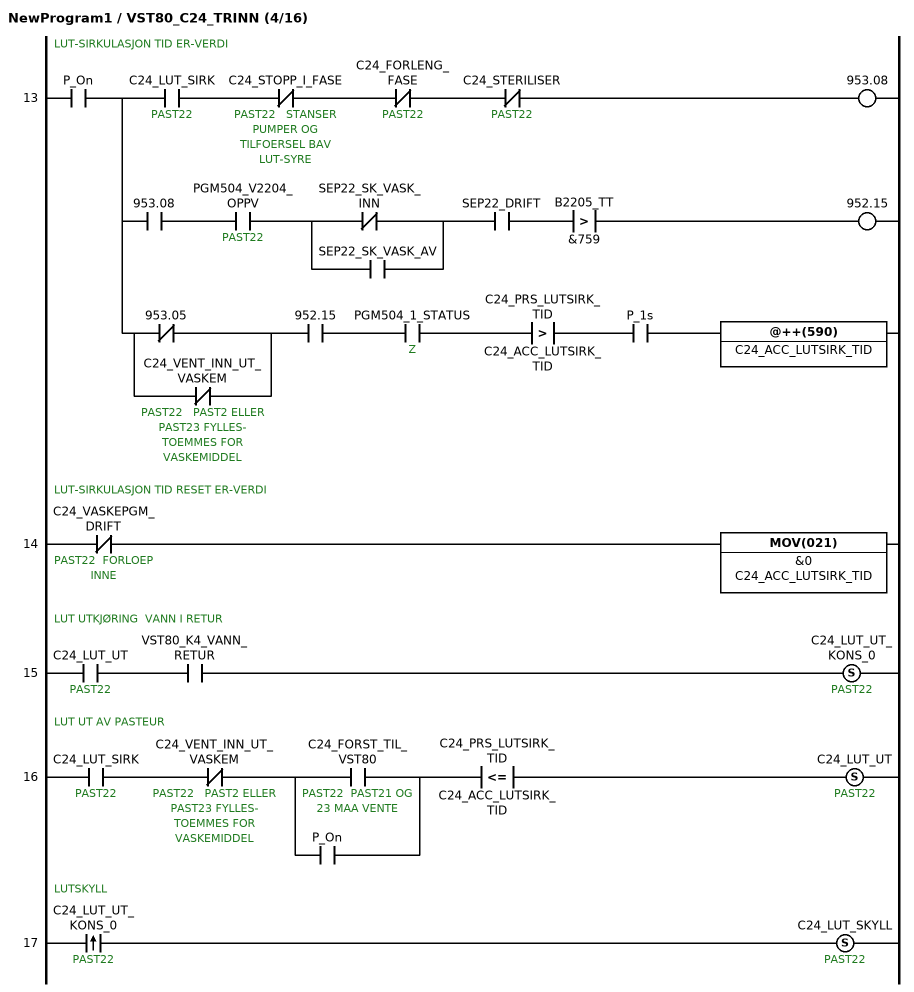
; [picture p432: NewProgram1 / VST80_C24_TRINN, rungs 13-17]
; rung 13: LUT-SIRKULASJON TID ER-VERDI
LD P_On
OUT TR0
AND C24_LUT_SIRK  ; PAST22
ANDNOT C24_STOPP_I_FASE  ; PAST22   STANSER PUMPER OG TILFOERSEL BAV LUT-SYRE
ANDNOT C24_FORLENG_FASE  ; PAST22
ANDNOT C24_STERILISER  ; PAST22
OUT 953.08
LD TR0
AND 953.08
AND PGM504_V2204_OPPV  ; PAST22
LDNOT SEP22_SK_VASK_INN
OR SEP22_SK_VASK_AV
ANDLD
AND SEP22_DRIFT
AND>(320) B2205_TT &759
OUT 952.15
LD TR0
LDNOT 953.05
ORNOT C24_VENT_INN_UT_VASKEM  ; PAST22   PAST2 ELLER PAST23 FYLLES-TOEMMES FOR VASKEMIDDEL
ANDLD
AND 952.15
AND PGM504_1_STATUS  ; Z
AND>(320) C24_PRS_LUTSIRK_TID C24_ACC_LUTSIRK_TID
AND P_1s
@++(590) C24_ACC_LUTSIRK_TID
; rung 14: LUT-SIRKULASJON TID RESET ER-VERDI
LDNOT C24_VASKEPGM_DRIFT  ; PAST22  FORLOEP INNE
MOV(021) &0 C24_ACC_LUTSIRK_TID
; rung 15: LUT UTKJØRING  VANN I RETUR
LD C24_LUT_UT  ; PAST22
AND VST80_K4_VANN_RETUR
SET C24_LUT_UT_KONS_0  ; PAST22
; rung 16: LUT UT AV PASTEUR
LD C24_LUT_SIRK  ; PAST22
ANDNOT C24_VENT_INN_UT_VASKEM  ; PAST22   PAST2 ELLER PAST23 FYLLES-TOEMMES FOR VASKEMIDDEL
LD C24_FORST_TIL_VST80  ; PAST22  PAST21 OG 23 MAA VENTE
OR P_On
ANDLD
AND<=(315) C24_PRS_LUTSIRK_TID C24_ACC_LUTSIRK_TID
SET C24_LUT_UT  ; PAST22
; rung 17: LUTSKYLL
@LD C24_LUT_UT_KONS_0  ; PAST22
SET C24_LUT_SKYLL  ; PAST22

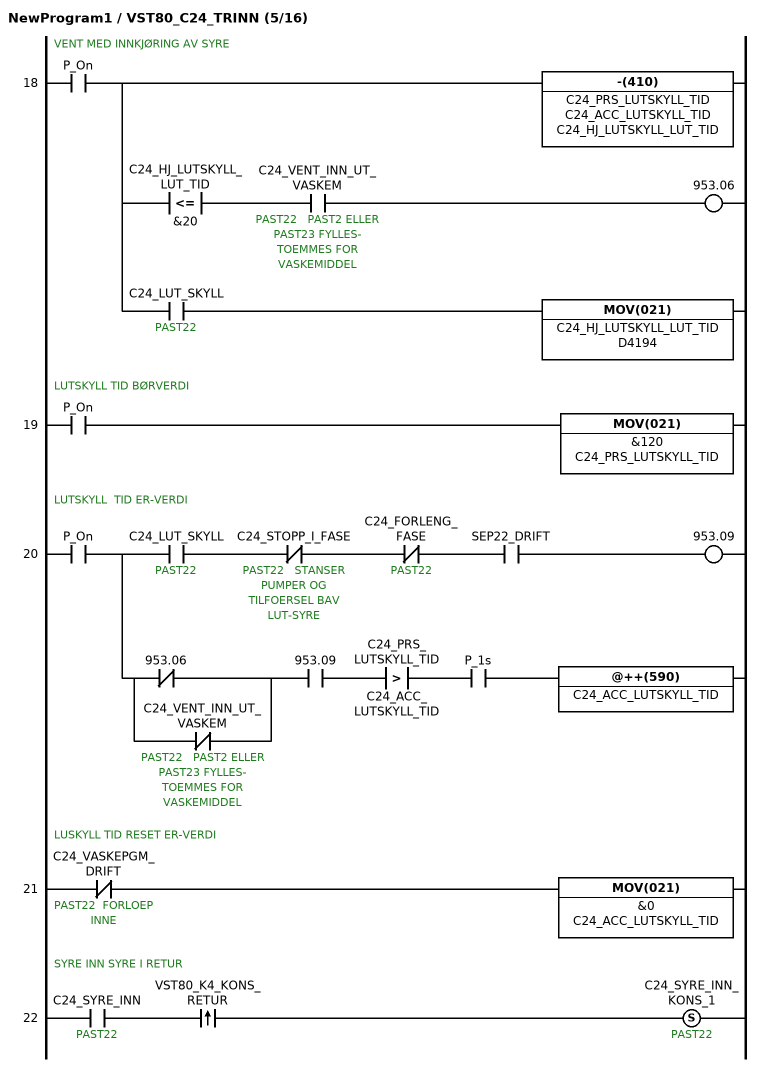
; rung 18: VENT MED INNKJØRING AV SYRE
LD P_On
OUT TR0
-(410) C24_PRS_LUTSKYLL_TID C24_ACC_LUTSKYLL_TID C24_HJ_LUTSKYLL_LUT_TID
AND<=(315) C24_HJ_LUTSKYLL_LUT_TID &20
AND C24_VENT_INN_UT_VASKEM  ; PAST22   PAST2 ELLER PAST23 FYLLES-TOEMMES FOR VASKEMIDDEL
OUT 953.06
LD TR0
AND C24_LUT_SKYLL  ; PAST22
MOV(021) C24_HJ_LUTSKYLL_LUT_TID D4194
; rung 19: LUTSKYLL TID BØRVERDI
LD P_On
MOV(021) &120 C24_PRS_LUTSKYLL_TID
; rung 20: LUTSKYLL  TID ER-VERDI
LD P_On
OUT TR0
AND C24_LUT_SKYLL  ; PAST22
ANDNOT C24_STOPP_I_FASE  ; PAST22   STANSER PUMPER OG TILFOERSEL BAV LUT-SYRE
ANDNOT C24_FORLENG_FASE  ; PAST22
AND SEP22_DRIFT
OUT 953.09
LD TR0
LDNOT 953.06
ORNOT C24_VENT_INN_UT_VASKEM  ; PAST22   PAST2 ELLER PAST23 FYLLES-TOEMMES FOR VASKEMIDDEL
ANDLD
AND 953.09
AND>(320) C24_PRS_LUTSKYLL_TID C24_ACC_LUTSKYLL_TID
AND P_1s
@++(590) C24_ACC_LUTSKYLL_TID
; rung 21: LUSKYLL TID RESET ER-VERDI
LDNOT C24_VASKEPGM_DRIFT  ; PAST22  FORLOEP INNE
MOV(021) &0 C24_ACC_LUTSKYLL_TID
; rung 22: SYRE INN SYRE I RETUR
LD C24_SYRE_INN  ; PAST22
@AND VST80_K4_KONS_RETUR
SET C24_SYRE_INN_KONS_1  ; PAST22

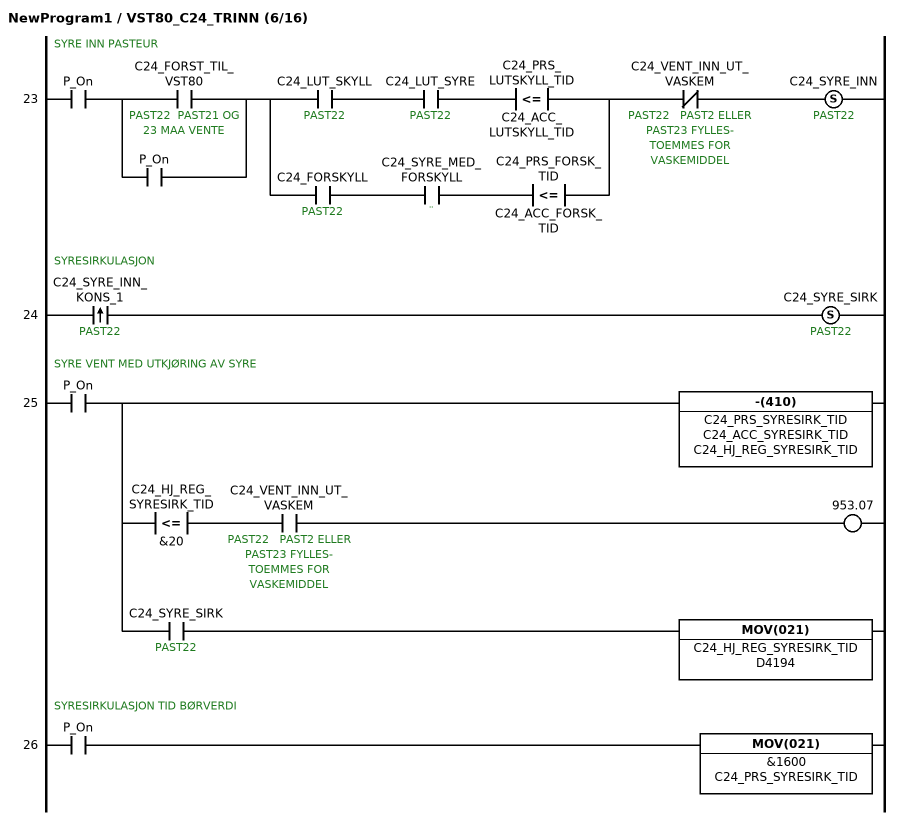
; rung 23: SYRE INN PASTEUR
LD P_On
LD C24_FORST_TIL_VST80  ; PAST22  PAST21 OG 23 MAA VENTE
OR P_On
ANDLD
LD C24_LUT_SKYLL  ; PAST22
AND C24_LUT_SYRE  ; PAST22
AND<=(315) C24_PRS_LUTSKYLL_TID C24_ACC_LUTSKYLL_TID
LD C24_FORSKYLL  ; PAST22
AND C24_SYRE_MED_FORSKYLL  ; ¨
AND<=(315) C24_PRS_FORSK_TID C24_ACC_FORSK_TID
ORLD
ANDLD
ANDNOT C24_VENT_INN_UT_VASKEM  ; PAST22   PAST2 ELLER PAST23 FYLLES-TOEMMES FOR VASKEMIDDEL
SET C24_SYRE_INN  ; PAST22
; rung 24: SYRESIRKULASJON
@LD C24_SYRE_INN_KONS_1  ; PAST22
SET C24_SYRE_SIRK  ; PAST22
; rung 25: SYRE VENT MED UTKJØRING AV SYRE
LD P_On
OUT TR0
-(410) C24_PRS_SYRESIRK_TID C24_ACC_SYRESIRK_TID C24_HJ_REG_SYRESIRK_TID
AND<=(315) C24_HJ_REG_SYRESIRK_TID &20
AND C24_VENT_INN_UT_VASKEM  ; PAST22   PAST2 ELLER PAST23 FYLLES-TOEMMES FOR VASKEMIDDEL
OUT 953.07
LD TR0
AND C24_SYRE_SIRK  ; PAST22
MOV(021) C24_HJ_REG_SYRESIRK_TID D4194
; rung 26: SYRESIRKULASJON TID BØRVERDI
LD P_On
MOV(021) &1600 C24_PRS_SYRESIRK_TID

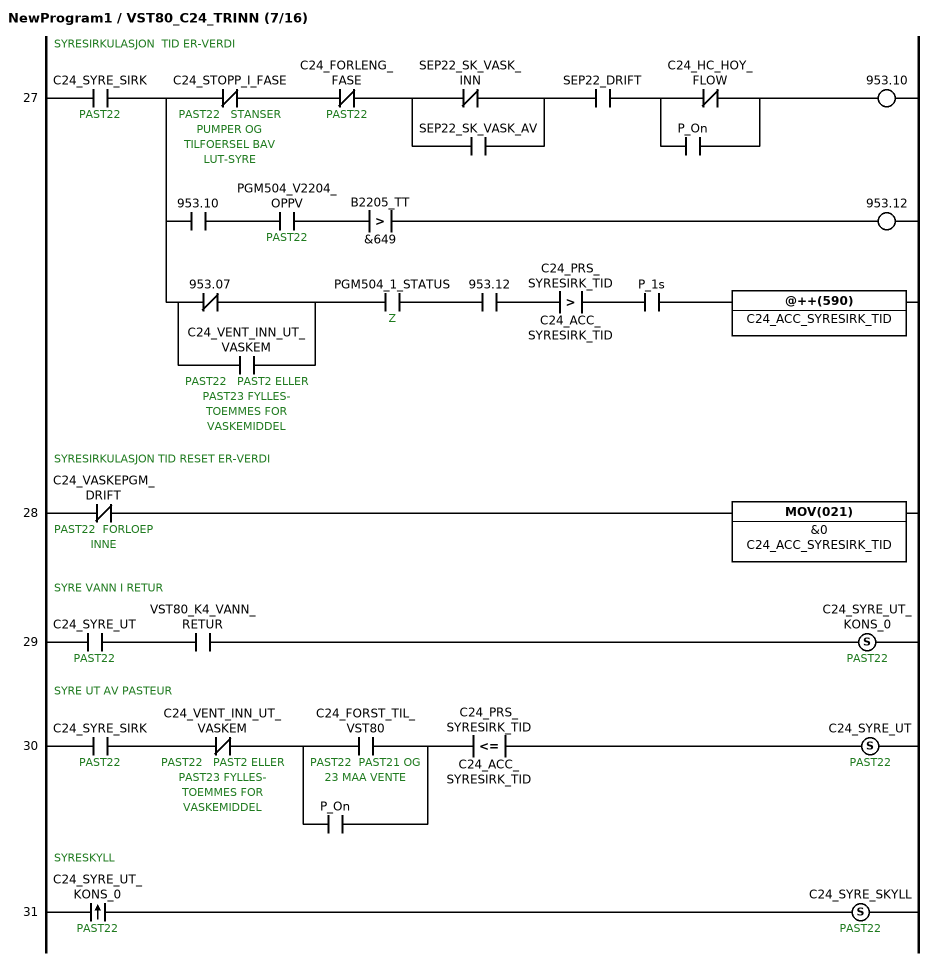
; rung 27: SYRESIRKULASJON  TID ER-VERDI
LD C24_SYRE_SIRK  ; PAST22
OUT TR0
ANDNOT C24_STOPP_I_FASE  ; PAST22   STANSER PUMPER OG TILFOERSEL BAV LUT-SYRE
ANDNOT C24_FORLENG_FASE  ; PAST22
LDNOT SEP22_SK_VASK_INN
OR SEP22_SK_VASK_AV
ANDLD
AND SEP22_DRIFT
LDNOT C24_HC_HOY_FLOW
OR P_On
ANDLD
OUT 953.10
LD TR0
AND 953.10
AND PGM504_V2204_OPPV  ; PAST22
AND>(320) B2205_TT &649
OUT 953.12
LD TR0
LDNOT 953.07
OR C24_VENT_INN_UT_VASKEM  ; PAST22   PAST2 ELLER PAST23 FYLLES-TOEMMES FOR VASKEMIDDEL
ANDLD
AND PGM504_1_STATUS  ; Z
AND 953.12
AND>(320) C24_PRS_SYRESIRK_TID C24_ACC_SYRESIRK_TID
AND P_1s
@++(590) C24_ACC_SYRESIRK_TID
; rung 28: SYRESIRKULASJON TID RESET ER-VERDI
LDNOT C24_VASKEPGM_DRIFT  ; PAST22  FORLOEP INNE
MOV(021) &0 C24_ACC_SYRESIRK_TID
; rung 29: SYRE VANN I RETUR
LD C24_SYRE_UT  ; PAST22
AND VST80_K4_VANN_RETUR
SET C24_SYRE_UT_KONS_0  ; PAST22
; rung 30: SYRE UT AV PASTEUR
LD C24_SYRE_SIRK  ; PAST22
ANDNOT C24_VENT_INN_UT_VASKEM  ; PAST22   PAST2 ELLER PAST23 FYLLES-TOEMMES FOR VASKEMIDDEL
LD C24_FORST_TIL_VST80  ; PAST22  PAST21 OG 23 MAA VENTE
OR P_On
ANDLD
AND<=(315) C24_PRS_SYRESIRK_TID C24_ACC_SYRESIRK_TID
SET C24_SYRE_UT  ; PAST22
; rung 31: SYRESKYLL
@LD C24_SYRE_UT_KONS_0  ; PAST22
SET C24_SYRE_SKYLL  ; PAST22

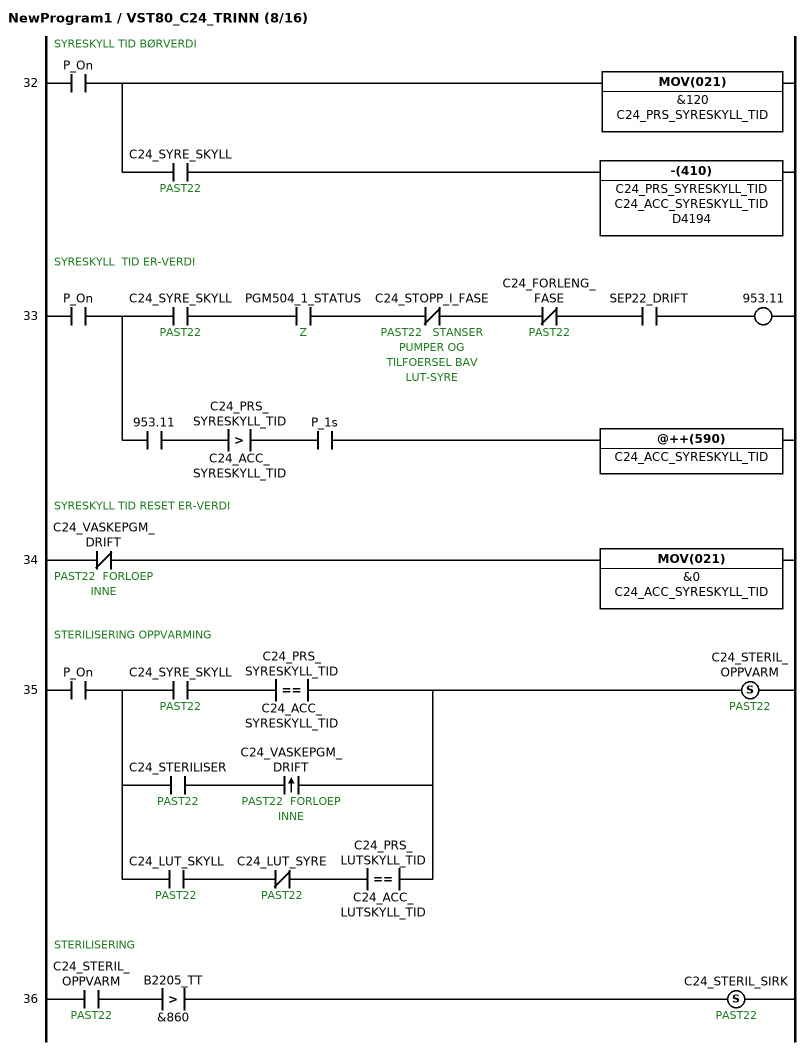
; rung 32: SYRESKYLL TID BØRVERDI
LD P_On
MOV(021) &120 C24_PRS_SYRESKYLL_TID
AND C24_SYRE_SKYLL  ; PAST22
-(410) C24_PRS_SYRESKYLL_TID C24_ACC_SYRESKYLL_TID D4194
; rung 33: SYRESKYLL  TID ER-VERDI
LD P_On
OUT TR0
AND C24_SYRE_SKYLL  ; PAST22
AND PGM504_1_STATUS  ; Z
ANDNOT C24_STOPP_I_FASE  ; PAST22   STANSER PUMPER OG TILFOERSEL BAV LUT-SYRE
ANDNOT C24_FORLENG_FASE  ; PAST22
AND SEP22_DRIFT
OUT 953.11
LD TR0
AND 953.11
AND>(320) C24_PRS_SYRESKYLL_TID C24_ACC_SYRESKYLL_TID
AND P_1s
@++(590) C24_ACC_SYRESKYLL_TID
; rung 34: SYRESKYLL TID RESET ER-VERDI
LDNOT C24_VASKEPGM_DRIFT  ; PAST22  FORLOEP INNE
MOV(021) &0 C24_ACC_SYRESKYLL_TID
; rung 35: STERILISERING OPPVARMING
LD P_On
LD C24_SYRE_SKYLL  ; PAST22
AND=(300) C24_PRS_SYRESKYLL_TID C24_ACC_SYRESKYLL_TID
LD C24_STERILISER  ; PAST22
@AND C24_VASKEPGM_DRIFT  ; PAST22  FORLOEP INNE
ORLD
LD C24_LUT_SKYLL  ; PAST22
ANDNOT C24_LUT_SYRE  ; PAST22
AND=(300) C24_PRS_LUTSKYLL_TID C24_ACC_LUTSKYLL_TID
ORLD
ANDLD
SET C24_STERIL_OPPVARM  ; PAST22
; rung 36: STERILISERING
LD C24_STERIL_OPPVARM  ; PAST22
AND>(320) B2205_TT &860
SET C24_STERIL_SIRK  ; PAST22

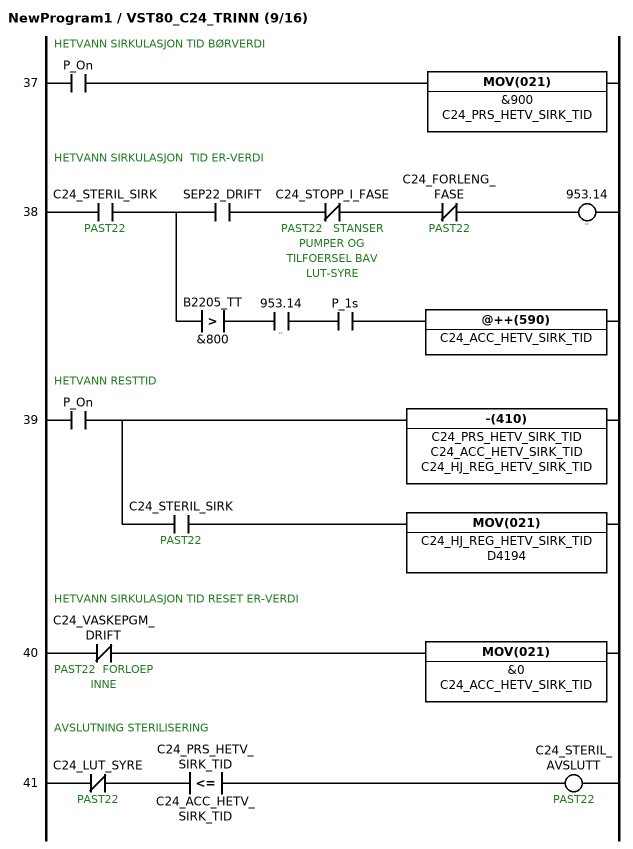
; rung 37: HETVANN SIRKULASJON TID BØRVERDI
LD P_On
MOV(021) &900 C24_PRS_HETV_SIRK_TID
; rung 38: HETVANN SIRKULASJON  TID ER-VERDI
LD C24_STERIL_SIRK  ; PAST22
OUT TR0
AND SEP22_DRIFT
ANDNOT C24_STOPP_I_FASE  ; PAST22   STANSER PUMPER OG TILFOERSEL BAV LUT-SYRE
ANDNOT C24_FORLENG_FASE  ; PAST22
OUT 953.14  ; ¨
LD TR0
AND>(320) B2205_TT &800
AND 953.14  ; ¨
AND P_1s
@++(590) C24_ACC_HETV_SIRK_TID
; rung 39: HETVANN RESTTID
LD P_On
-(410) C24_PRS_HETV_SIRK_TID C24_ACC_HETV_SIRK_TID C24_HJ_REG_HETV_SIRK_TID
AND C24_STERIL_SIRK  ; PAST22
MOV(021) C24_HJ_REG_HETV_SIRK_TID D4194
; rung 40: HETVANN SIRKULASJON TID RESET ER-VERDI
LDNOT C24_VASKEPGM_DRIFT  ; PAST22  FORLOEP INNE
MOV(021) &0 C24_ACC_HETV_SIRK_TID
; rung 41: AVSLUTNING STERILISERING
LDNOT C24_LUT_SYRE  ; PAST22
AND<=(315) C24_PRS_HETV_SIRK_TID C24_ACC_HETV_SIRK_TID
OUT C24_STERIL_AVSLUTT  ; PAST22

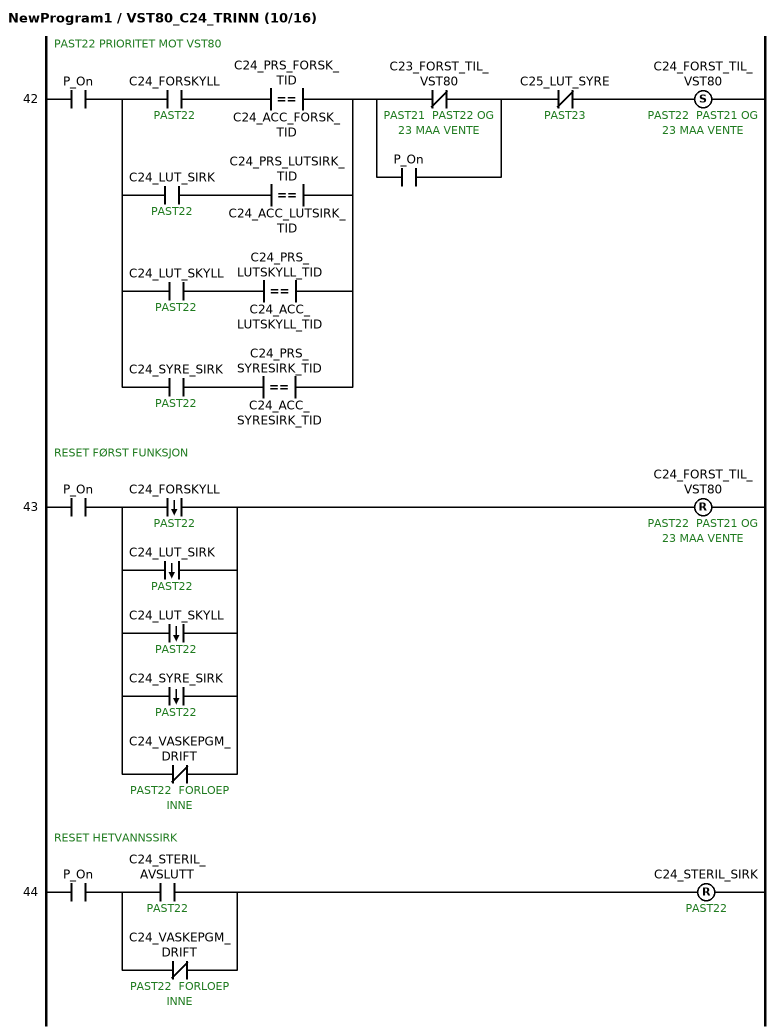
; rung 42: PAST22 PRIORITET MOT VST80
LD P_On
LD C24_FORSKYLL  ; PAST22
AND=(300) C24_PRS_FORSK_TID C24_ACC_FORSK_TID
LD C24_LUT_SIRK  ; PAST22
AND=(300) C24_PRS_LUTSIRK_TID C24_ACC_LUTSIRK_TID
ORLD
LD C24_LUT_SKYLL  ; PAST22
AND=(300) C24_PRS_LUTSKYLL_TID C24_ACC_LUTSKYLL_TID
ORLD
LD C24_SYRE_SIRK  ; PAST22
AND=(300) C24_PRS_SYRESIRK_TID C24_ACC_SYRESIRK_TID
ORLD
ANDLD
LDNOT C23_FORST_TIL_VST80  ; PAST21  PAST22 OG 23 MAA VENTE
OR P_On
ANDLD
ANDNOT C25_LUT_SYRE  ; PAST23
SET C24_FORST_TIL_VST80  ; PAST22  PAST21 OG 23 MAA VENTE
; rung 43: RESET FØRST FUNKSJON
LD P_On
%LD C24_FORSKYLL  ; PAST22
%OR C24_LUT_SIRK  ; PAST22
%OR C24_LUT_SKYLL  ; PAST22
%OR C24_SYRE_SIRK  ; PAST22
ORNOT C24_VASKEPGM_DRIFT  ; PAST22  FORLOEP INNE
ANDLD
RSET C24_FORST_TIL_VST80  ; PAST22  PAST21 OG 23 MAA VENTE
; rung 44: RESET HETVANNSSIRK
LD P_On
LD C24_STERIL_AVSLUTT  ; PAST22
ORNOT C24_VASKEPGM_DRIFT  ; PAST22  FORLOEP INNE
ANDLD
RSET C24_STERIL_SIRK  ; PAST22

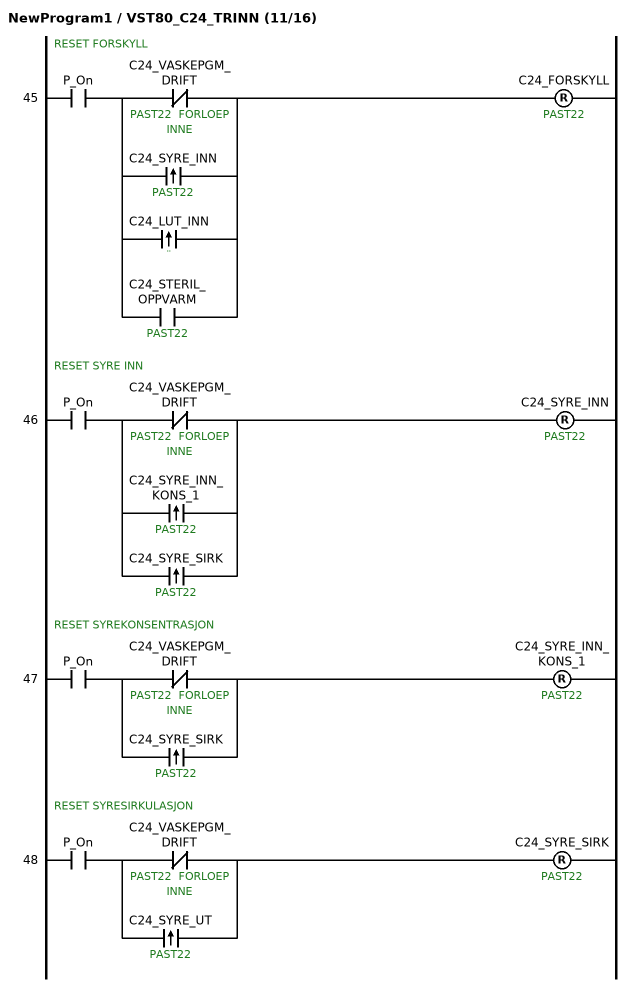
; rung 45: RESET FORSKYLL
LD P_On
LDNOT C24_VASKEPGM_DRIFT  ; PAST22  FORLOEP INNE
@OR C24_SYRE_INN  ; PAST22
@OR C24_LUT_INN  ; ¨
OR C24_STERIL_OPPVARM  ; PAST22
ANDLD
RSET C24_FORSKYLL  ; PAST22
; rung 46: RESET SYRE INN
LD P_On
LDNOT C24_VASKEPGM_DRIFT  ; PAST22  FORLOEP INNE
@OR C24_SYRE_INN_KONS_1  ; PAST22
@OR C24_SYRE_SIRK  ; PAST22
ANDLD
RSET C24_SYRE_INN  ; PAST22
; rung 47: RESET SYREKONSENTRASJON
LD P_On
LDNOT C24_VASKEPGM_DRIFT  ; PAST22  FORLOEP INNE
@OR C24_SYRE_SIRK  ; PAST22
ANDLD
RSET C24_SYRE_INN_KONS_1  ; PAST22
; rung 48: RESET SYRESIRKULASJON
LD P_On
LDNOT C24_VASKEPGM_DRIFT  ; PAST22  FORLOEP INNE
@OR C24_SYRE_UT  ; PAST22
ANDLD
RSET C24_SYRE_SIRK  ; PAST22

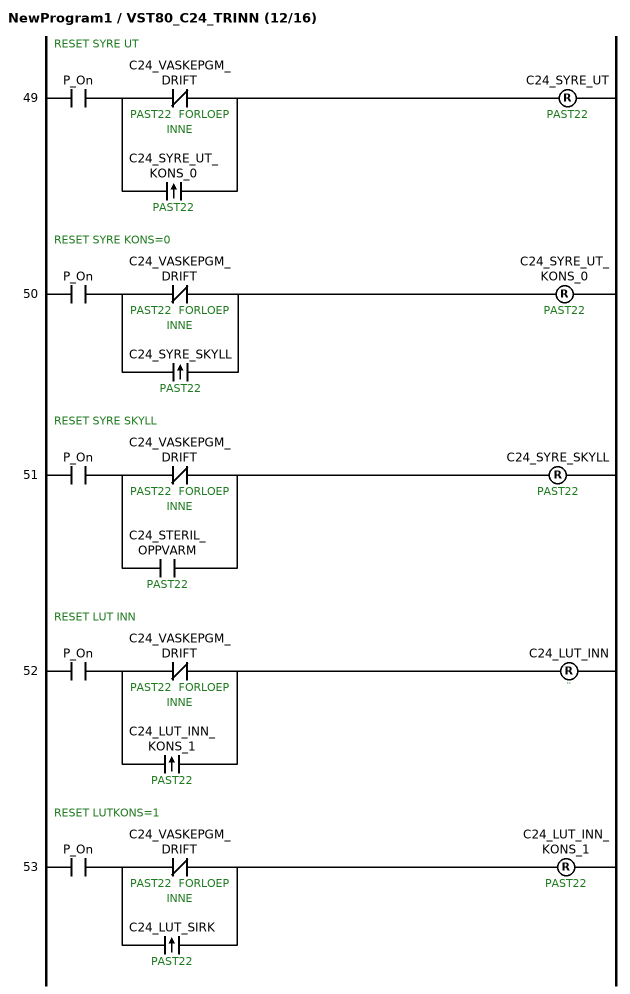
; rung 49: RESET SYRE UT
LD P_On
LDNOT C24_VASKEPGM_DRIFT  ; PAST22  FORLOEP INNE
@OR C24_SYRE_UT_KONS_0  ; PAST22
ANDLD
RSET C24_SYRE_UT  ; PAST22
; rung 50: RESET SYRE KONS=0
LD P_On
LDNOT C24_VASKEPGM_DRIFT  ; PAST22  FORLOEP INNE
@OR C24_SYRE_SKYLL  ; PAST22
ANDLD
RSET C24_SYRE_UT_KONS_0  ; PAST22
; rung 51: RESET SYRE SKYLL
LD P_On
LDNOT C24_VASKEPGM_DRIFT  ; PAST22  FORLOEP INNE
OR C24_STERIL_OPPVARM  ; PAST22
ANDLD
RSET C24_SYRE_SKYLL  ; PAST22
; rung 52: RESET LUT INN
LD P_On
LDNOT C24_VASKEPGM_DRIFT  ; PAST22  FORLOEP INNE
@OR C24_LUT_INN_KONS_1  ; PAST22
ANDLD
RSET C24_LUT_INN  ; ¨
; rung 53: RESET LUTKONS=1
LD P_On
LDNOT C24_VASKEPGM_DRIFT  ; PAST22  FORLOEP INNE
@OR C24_LUT_SIRK  ; PAST22
ANDLD
RSET C24_LUT_INN_KONS_1  ; PAST22

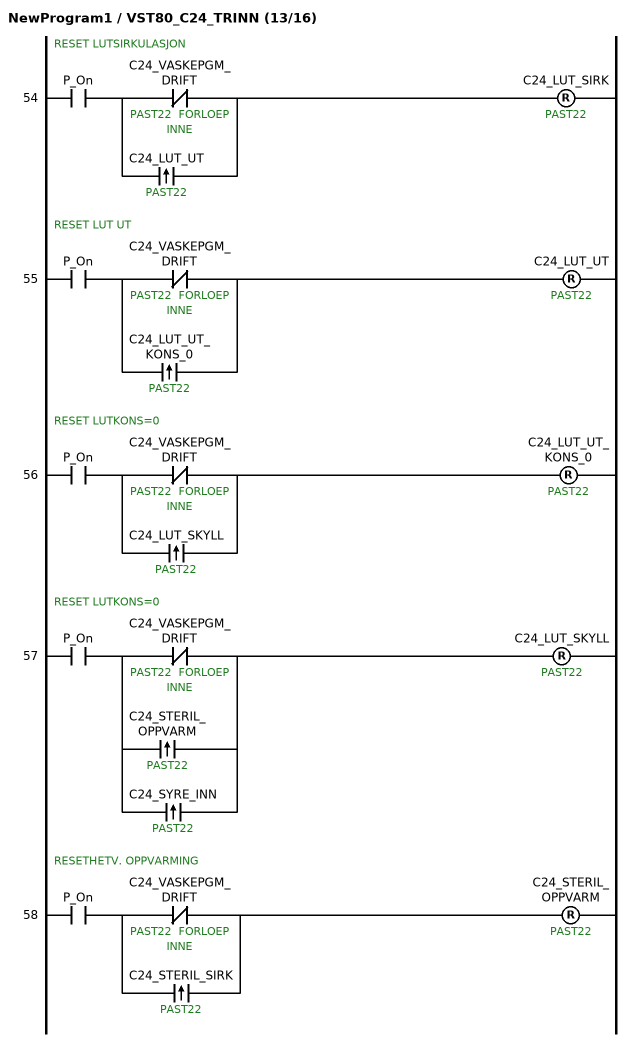
; rung 54: RESET LUTSIRKULASJON
LD P_On
LDNOT C24_VASKEPGM_DRIFT  ; PAST22  FORLOEP INNE
@OR C24_LUT_UT  ; PAST22
ANDLD
RSET C24_LUT_SIRK  ; PAST22
; rung 55: RESET LUT UT
LD P_On
LDNOT C24_VASKEPGM_DRIFT  ; PAST22  FORLOEP INNE
@OR C24_LUT_UT_KONS_0  ; PAST22
ANDLD
RSET C24_LUT_UT  ; PAST22
; rung 56: RESET LUTKONS=0
LD P_On
LDNOT C24_VASKEPGM_DRIFT  ; PAST22  FORLOEP INNE
@OR C24_LUT_SKYLL  ; PAST22
ANDLD
RSET C24_LUT_UT_KONS_0  ; PAST22
; rung 57: RESET LUTKONS=0
LD P_On
LDNOT C24_VASKEPGM_DRIFT  ; PAST22  FORLOEP INNE
@OR C24_STERIL_OPPVARM  ; PAST22
@OR C24_SYRE_INN  ; PAST22
ANDLD
RSET C24_LUT_SKYLL  ; PAST22
; rung 58: RESETHETV. OPPVARMING
LD P_On
LDNOT C24_VASKEPGM_DRIFT  ; PAST22  FORLOEP INNE
@OR C24_STERIL_SIRK  ; PAST22
ANDLD
RSET C24_STERIL_OPPVARM  ; PAST22

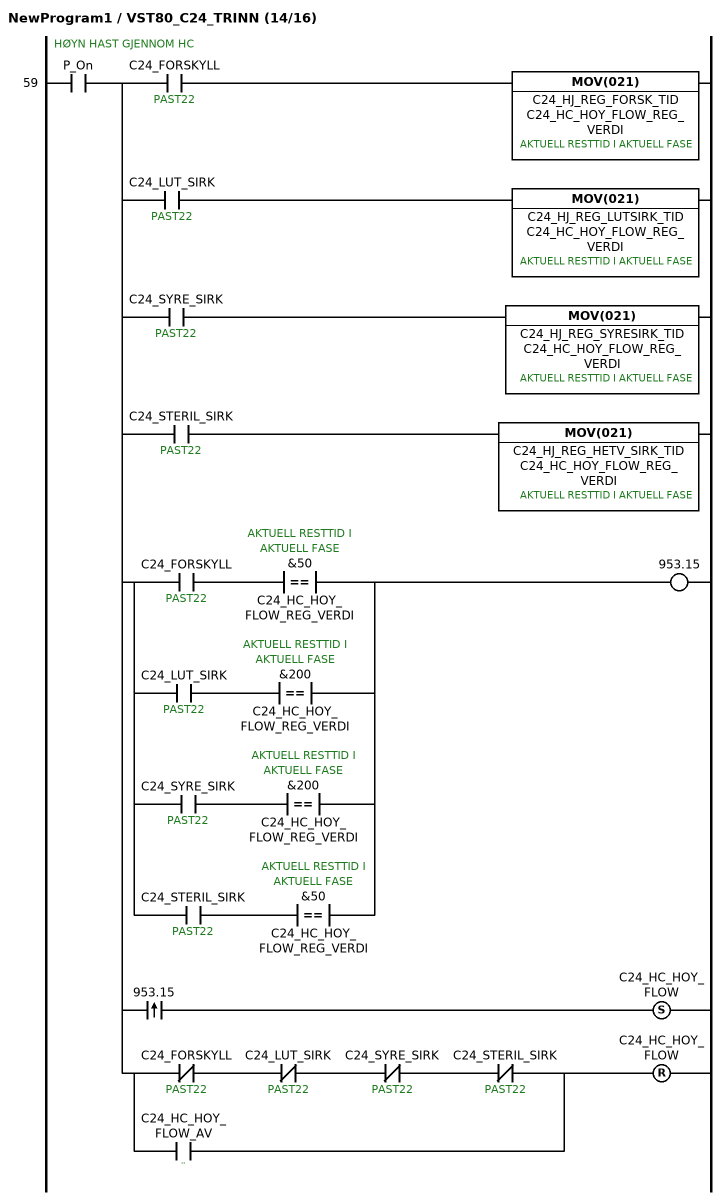
; rung 59: HØYN HAST GJENNOM HC
LD P_On
OUT TR0
AND C24_FORSKYLL  ; PAST22
MOV(021) C24_HJ_REG_FORSK_TID C24_HC_HOY_FLOW_REG_VERDI  ; AKTUELL RESTTID I AKTUELL FASE
LD TR0
AND C24_LUT_SIRK  ; PAST22
MOV(021) C24_HJ_REG_LUTSIRK_TID C24_HC_HOY_FLOW_REG_VERDI  ; AKTUELL RESTTID I AKTUELL FASE
LD TR0
AND C24_SYRE_SIRK  ; PAST22
MOV(021) C24_HJ_REG_SYRESIRK_TID C24_HC_HOY_FLOW_REG_VERDI  ; AKTUELL RESTTID I AKTUELL FASE
LD TR0
AND C24_STERIL_SIRK  ; PAST22
MOV(021) C24_HJ_REG_HETV_SIRK_TID C24_HC_HOY_FLOW_REG_VERDI  ; AKTUELL RESTTID I AKTUELL FASE
LD TR0
LD C24_FORSKYLL  ; PAST22
AND=(300) &50 C24_HC_HOY_FLOW_REG_VERDI  ; AKTUELL RESTTID I AKTUELL FASE
LD C24_LUT_SIRK  ; PAST22
AND=(300) &200 C24_HC_HOY_FLOW_REG_VERDI  ; AKTUELL RESTTID I AKTUELL FASE
ORLD
LD C24_SYRE_SIRK  ; PAST22
AND=(300) &200 C24_HC_HOY_FLOW_REG_VERDI  ; AKTUELL RESTTID I AKTUELL FASE
ORLD
LD C24_STERIL_SIRK  ; PAST22
AND=(300) &50 C24_HC_HOY_FLOW_REG_VERDI  ; AKTUELL RESTTID I AKTUELL FASE
ORLD
ANDLD
OUT 953.15
LD TR0
@AND 953.15
SET C24_HC_HOY_FLOW
LD TR0
LDNOT C24_FORSKYLL  ; PAST22
ANDNOT C24_LUT_SIRK  ; PAST22
ANDNOT C24_SYRE_SIRK  ; PAST22
ANDNOT C24_STERIL_SIRK  ; PAST22
OR C24_HC_HOY_FLOW_AV  ; ¨
ANDLD
RSET C24_HC_HOY_FLOW

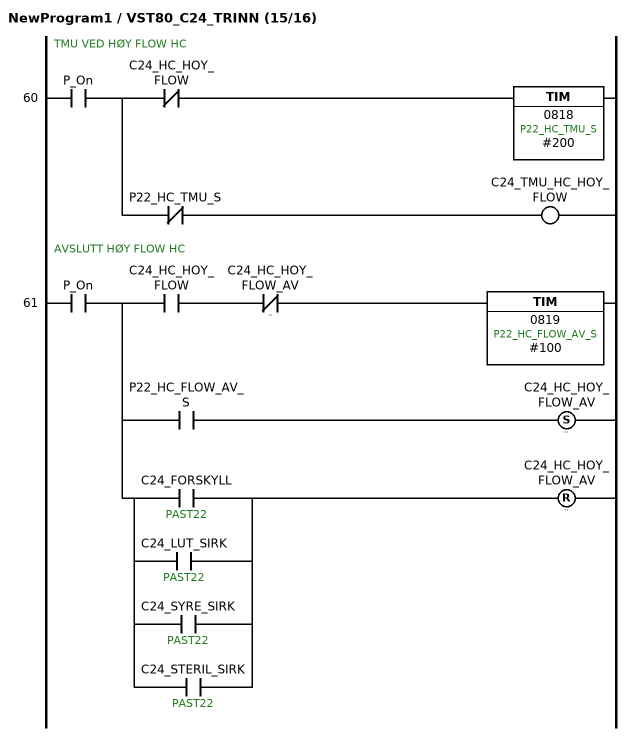
; rung 60: TMU VED HØY FLOW HC
LD P_On
OUT TR0
ANDNOT C24_HC_HOY_FLOW
TIM 0818 #200  ; P22_HC_TMU_S
LD TR0
ANDNOT P22_HC_TMU_S
OUT C24_TMU_HC_HOY_FLOW
; rung 61: AVSLUTT HØY FLOW HC
LD P_On
OUT TR0
AND C24_HC_HOY_FLOW
ANDNOT C24_HC_HOY_FLOW_AV  ; ¨
TIM 0819 #100  ; P22_HC_FLOW_AV_S
LD TR0
AND P22_HC_FLOW_AV_S
SET C24_HC_HOY_FLOW_AV  ; ¨
LD TR0
LD C24_FORSKYLL  ; PAST22
OR C24_LUT_SIRK  ; PAST22
OR C24_SYRE_SIRK  ; PAST22
OR C24_STERIL_SIRK  ; PAST22
ANDLD
RSET C24_HC_HOY_FLOW_AV  ; ¨

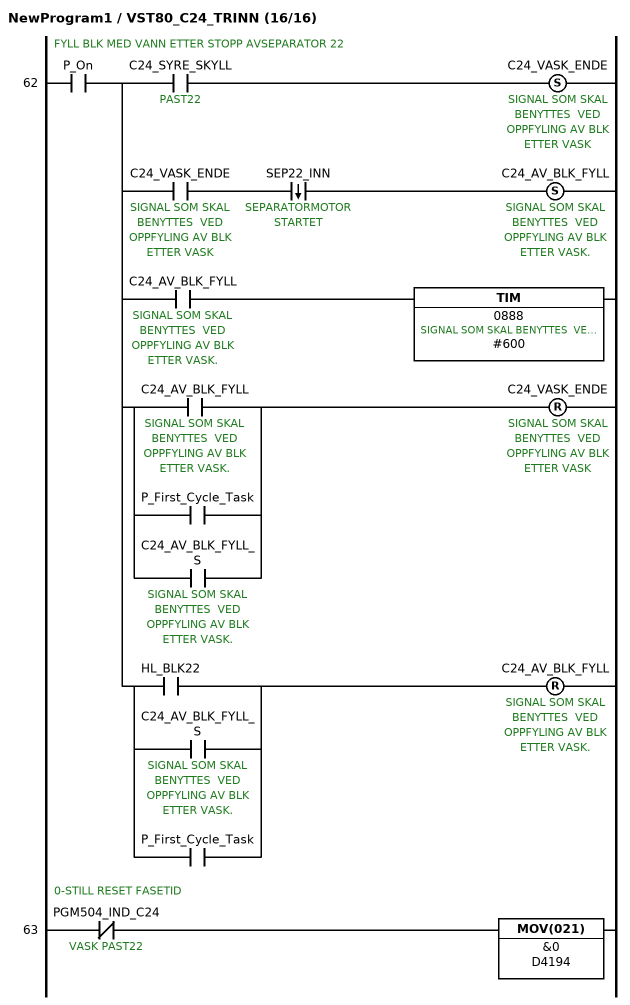
; rung 62: FYLL BLK MED VANN ETTER STOPP AVSEPARATOR 22
LD P_On
OUT TR0
AND C24_SYRE_SKYLL  ; PAST22
SET C24_VASK_ENDE  ; SIGNAL SOM SKAL BENYTTES  VED OPPFYLING AV BLK ETTER VASK
LD TR0
AND C24_VASK_ENDE  ; SIGNAL SOM SKAL BENYTTES  VED OPPFYLING AV BLK ETTER VASK
%AND SEP22_INN  ; SEPARATORMOTOR STARTET
SET C24_AV_BLK_FYLL  ; SIGNAL SOM SKAL BENYTTES  VED OPPFYLING AV BLK ETTER VASK.
LD TR0
AND C24_AV_BLK_FYLL  ; SIGNAL SOM SKAL BENYTTES  VED OPPFYLING AV BLK ETTER VASK.
TIM 0888 #600  ; SIGNAL SOM SKAL BENYTTES  VED OPPFYLING AV BLK ETTER VASK.
LD TR0
LD C24_AV_BLK_FYLL  ; SIGNAL SOM SKAL BENYTTES  VED OPPFYLING AV BLK ETTER VASK.
OR P_First_Cycle_Task
OR C24_AV_BLK_FYLL_S  ; SIGNAL SOM SKAL BENYTTES  VED OPPFYLING AV BLK ETTER VASK.
ANDLD
RSET C24_VASK_ENDE  ; SIGNAL SOM SKAL BENYTTES  VED OPPFYLING AV BLK ETTER VASK
LD TR0
LD HL_BLK22
OR C24_AV_BLK_FYLL_S  ; SIGNAL SOM SKAL BENYTTES  VED OPPFYLING AV BLK ETTER VASK.
OR P_First_Cycle_Task
ANDLD
RSET C24_AV_BLK_FYLL  ; SIGNAL SOM SKAL BENYTTES  VED OPPFYLING AV BLK ETTER VASK.
; rung 63: 0-STILL RESET FASETID
LDNOT PGM504_IND_C24  ; VASK PAST22
MOV(021) &0 D4194
; rung 64: Ingen_kommentar_funnet

### Section VST80_C24_GRAFIKK_TEKSTER

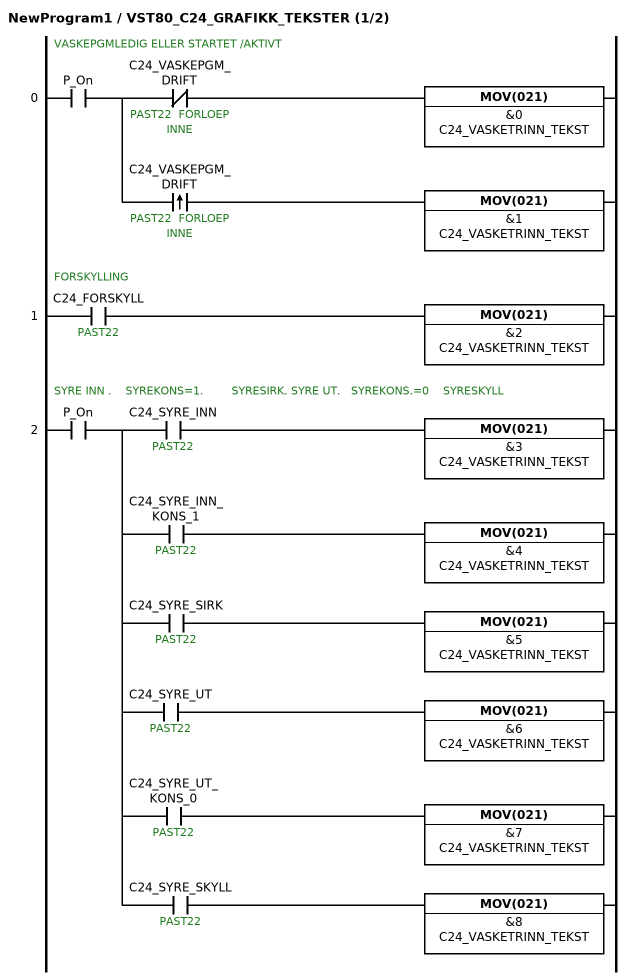
; rung 0: VASKEPGMLEDIG ELLER STARTET /AKTIVT
LD P_On
OUT TR0
ANDNOT C24_VASKEPGM_DRIFT  ; PAST22  FORLOEP INNE
MOV(021) &0 C24_VASKETRINN_TEKST
LD TR0
@AND C24_VASKEPGM_DRIFT  ; PAST22  FORLOEP INNE
MOV(021) &1 C24_VASKETRINN_TEKST
; rung 1: FORSKYLLING
LD C24_FORSKYLL  ; PAST22
MOV(021) &2 C24_VASKETRINN_TEKST
; rung 2: SYRE INN .    SYREKONS=1.        SYRESIRK. SYRE UT.   SYREKONS.=0    SYRESKYLL
LD P_On
OUT TR0
AND C24_SYRE_INN  ; PAST22
MOV(021) &3 C24_VASKETRINN_TEKST
LD TR0
AND C24_SYRE_INN_KONS_1  ; PAST22
MOV(021) &4 C24_VASKETRINN_TEKST
LD TR0
AND C24_SYRE_SIRK  ; PAST22
MOV(021) &5 C24_VASKETRINN_TEKST
LD TR0
AND C24_SYRE_UT  ; PAST22
MOV(021) &6 C24_VASKETRINN_TEKST
LD TR0
AND C24_SYRE_UT_KONS_0  ; PAST22
MOV(021) &7 C24_VASKETRINN_TEKST
LD TR0
AND C24_SYRE_SKYLL  ; PAST22
MOV(021) &8 C24_VASKETRINN_TEKST

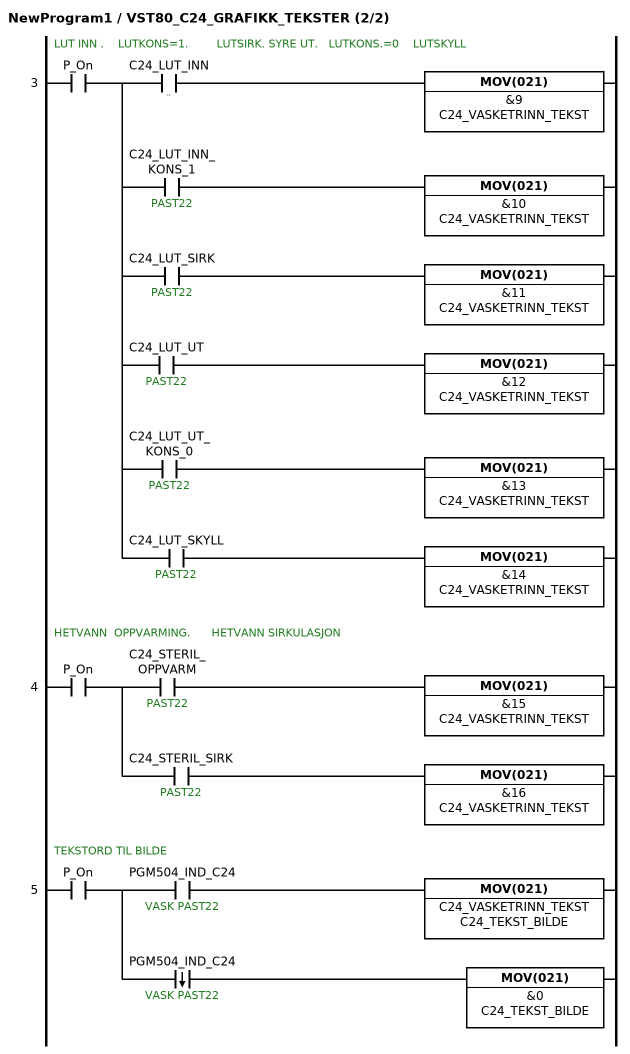
; rung 3: LUT INN .    LUTKONS=1.        LUTSIRK. SYRE UT.   LUTKONS.=0    LUTSKYLL
LD P_On
OUT TR0
AND C24_LUT_INN  ; ¨
MOV(021) &9 C24_VASKETRINN_TEKST
LD TR0
AND C24_LUT_INN_KONS_1  ; PAST22
MOV(021) &10 C24_VASKETRINN_TEKST
LD TR0
AND C24_LUT_SIRK  ; PAST22
MOV(021) &11 C24_VASKETRINN_TEKST
LD TR0
AND C24_LUT_UT  ; PAST22
MOV(021) &12 C24_VASKETRINN_TEKST
LD TR0
AND C24_LUT_UT_KONS_0  ; PAST22
MOV(021) &13 C24_VASKETRINN_TEKST
LD TR0
AND C24_LUT_SKYLL  ; PAST22
MOV(021) &14 C24_VASKETRINN_TEKST
; rung 4: HETVANN  OPPVARMING.      HETVANN SIRKULASJON
LD P_On
OUT TR0
AND C24_STERIL_OPPVARM  ; PAST22
MOV(021) &15 C24_VASKETRINN_TEKST
LD TR0
AND C24_STERIL_SIRK  ; PAST22
MOV(021) &16 C24_VASKETRINN_TEKST
; rung 5: TEKSTORD TIL BILDE
LD P_On
OUT TR0
AND PGM504_IND_C24  ; VASK PAST22
MOV(021) C24_VASKETRINN_TEKST C24_TEKST_BILDE
LD TR0
%AND PGM504_IND_C24  ; VASK PAST22
MOV(021) &0 C24_TEKST_BILDE
; rung 6: Ingen_kommentar_funnet

### Section C24_VASKERAPORT

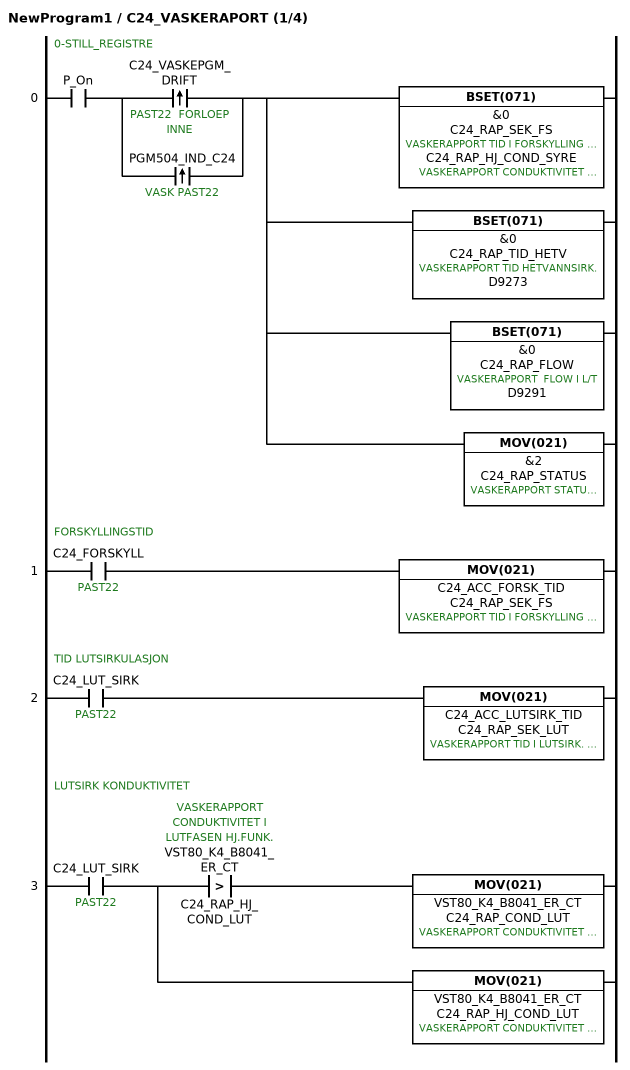
; rung 0: 0-STILL_REGISTRE
LD P_On
@LD C24_VASKEPGM_DRIFT  ; PAST22  FORLOEP INNE
@OR PGM504_IND_C24  ; VASK PAST22
ANDLD
BSET(071) &0 C24_RAP_SEK_FS C24_RAP_HJ_COND_SYRE  ; VASKERAPPORT TID I FORSKYLLING I SEKUNDER, VASKERAPPORT CONDUKTIVITET I SYREFASEN HJ.FUNK.
BSET(071) &0 C24_RAP_TID_HETV D9273  ; VASKERAPPORT TID HETVANNSIRK.
BSET(071) &0 C24_RAP_FLOW D9291  ; VASKERAPPORT  FLOW I L/T
MOV(021) &2 C24_RAP_STATUS  ; VASKERAPPORT STATUS          0=GODKJ.  1=DRIFTFORS.  2= IKKE GODKJ.
; rung 1: FORSKYLLINGSTID
LD C24_FORSKYLL  ; PAST22
MOV(021) C24_ACC_FORSK_TID C24_RAP_SEK_FS  ; VASKERAPPORT TID I FORSKYLLING I SEKUNDER
; rung 2: TID LUTSIRKULASJON
LD C24_LUT_SIRK  ; PAST22
MOV(021) C24_ACC_LUTSIRK_TID C24_RAP_SEK_LUT  ; VASKERAPPORT TID I LUTSIRK. I SEKUNDER
; rung 3: LUTSIRK KONDUKTIVITET
LD C24_LUT_SIRK  ; PAST22
OUT TR0
AND>(320) VST80_K4_B8041_ER_CT C24_RAP_HJ_COND_LUT  ; VASKERAPPORT CONDUKTIVITET I LUTFASEN HJ.FUNK.
MOV(021) VST80_K4_B8041_ER_CT C24_RAP_COND_LUT  ; VASKERAPPORT CONDUKTIVITET I LUTFASEN
LD TR0
MOV(021) VST80_K4_B8041_ER_CT C24_RAP_HJ_COND_LUT  ; VASKERAPPORT CONDUKTIVITET I LUTFASEN HJ.FUNK.

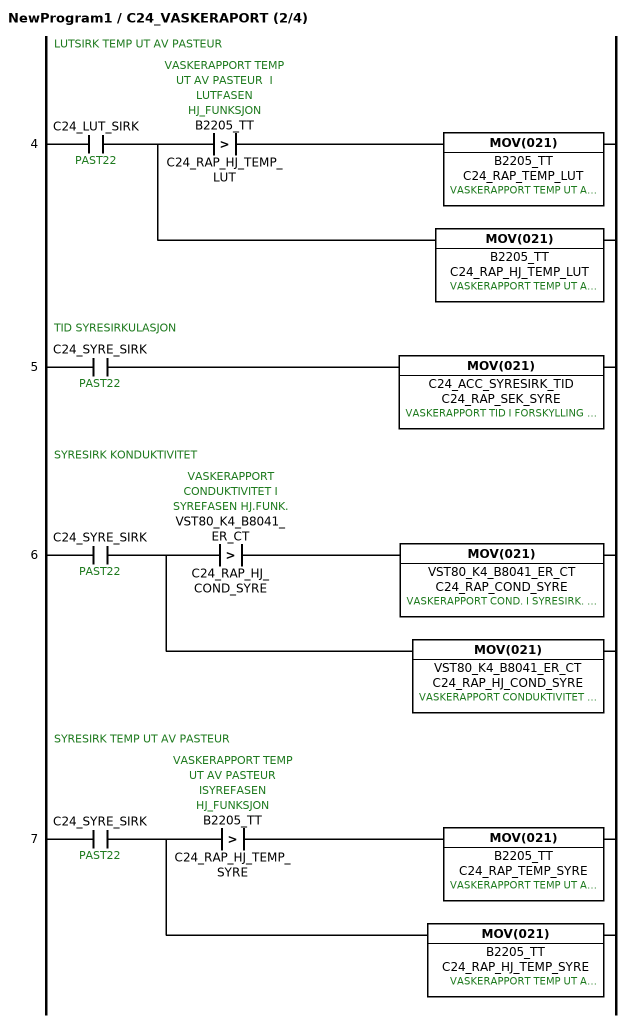
; rung 4: LUTSIRK TEMP UT AV PASTEUR
LD C24_LUT_SIRK  ; PAST22
OUT TR0
AND>(320) B2205_TT C24_RAP_HJ_TEMP_LUT  ; VASKERAPPORT TEMP UT AV PASTEUR  I LUTFASEN HJ_FUNKSJON
MOV(021) B2205_TT C24_RAP_TEMP_LUT  ; VASKERAPPORT TEMP UT AV PASTEUR  I LUTFASEN
LD TR0
MOV(021) B2205_TT C24_RAP_HJ_TEMP_LUT  ; VASKERAPPORT TEMP UT AV PASTEUR  I LUTFASEN HJ_FUNKSJON
; rung 5: TID SYRESIRKULASJON
LD C24_SYRE_SIRK  ; PAST22
MOV(021) C24_ACC_SYRESIRK_TID C24_RAP_SEK_SYRE  ; VASKERAPPORT TID I FORSKYLLING I SEKUNDER
; rung 6: SYRESIRK KONDUKTIVITET
LD C24_SYRE_SIRK  ; PAST22
OUT TR0
AND>(320) VST80_K4_B8041_ER_CT C24_RAP_HJ_COND_SYRE  ; VASKERAPPORT CONDUKTIVITET I SYREFASEN HJ.FUNK.
MOV(021) VST80_K4_B8041_ER_CT C24_RAP_COND_SYRE  ; VASKERAPPORT COND. I SYRESIRK. I SEKUNDER
LD TR0
MOV(021) VST80_K4_B8041_ER_CT C24_RAP_HJ_COND_SYRE  ; VASKERAPPORT CONDUKTIVITET I SYREFASEN HJ.FUNK.
; rung 7: SYRESIRK TEMP UT AV PASTEUR
LD C24_SYRE_SIRK  ; PAST22
OUT TR0
AND>(320) B2205_TT C24_RAP_HJ_TEMP_SYRE  ; VASKERAPPORT TEMP UT AV PASTEUR ISYREFASEN HJ_FUNKSJON
MOV(021) B2205_TT C24_RAP_TEMP_SYRE  ; VASKERAPPORT TEMP UT AV PASTEUR ISYREFASEN
LD TR0
MOV(021) B2205_TT C24_RAP_HJ_TEMP_SYRE  ; VASKERAPPORT TEMP UT AV PASTEUR ISYREFASEN HJ_FUNKSJON

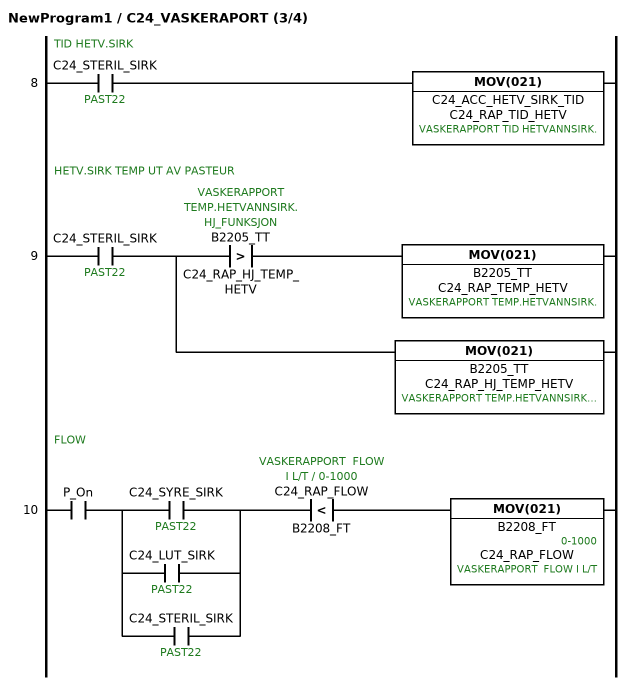
; rung 8: TID HETV.SIRK
LD C24_STERIL_SIRK  ; PAST22
MOV(021) C24_ACC_HETV_SIRK_TID C24_RAP_TID_HETV  ; VASKERAPPORT TID HETVANNSIRK.
; rung 9: HETV.SIRK TEMP UT AV PASTEUR
LD C24_STERIL_SIRK  ; PAST22
OUT TR0
AND>(320) B2205_TT C24_RAP_HJ_TEMP_HETV  ; VASKERAPPORT TEMP.HETVANNSIRK. HJ_FUNKSJON
MOV(021) B2205_TT C24_RAP_TEMP_HETV  ; VASKERAPPORT TEMP.HETVANNSIRK.
LD TR0
MOV(021) B2205_TT C24_RAP_HJ_TEMP_HETV  ; VASKERAPPORT TEMP.HETVANNSIRK. HJ_FUNKSJON
; rung 10: FLOW
LD P_On
LD C24_SYRE_SIRK  ; PAST22
OR C24_LUT_SIRK  ; PAST22
OR C24_STERIL_SIRK  ; PAST22
ANDLD
AND<(310) C24_RAP_FLOW B2208_FT  ; VASKERAPPORT  FLOW I L/T, 0-1000
MOV(021) B2208_FT C24_RAP_FLOW  ; 0-1000, VASKERAPPORT  FLOW I L/T

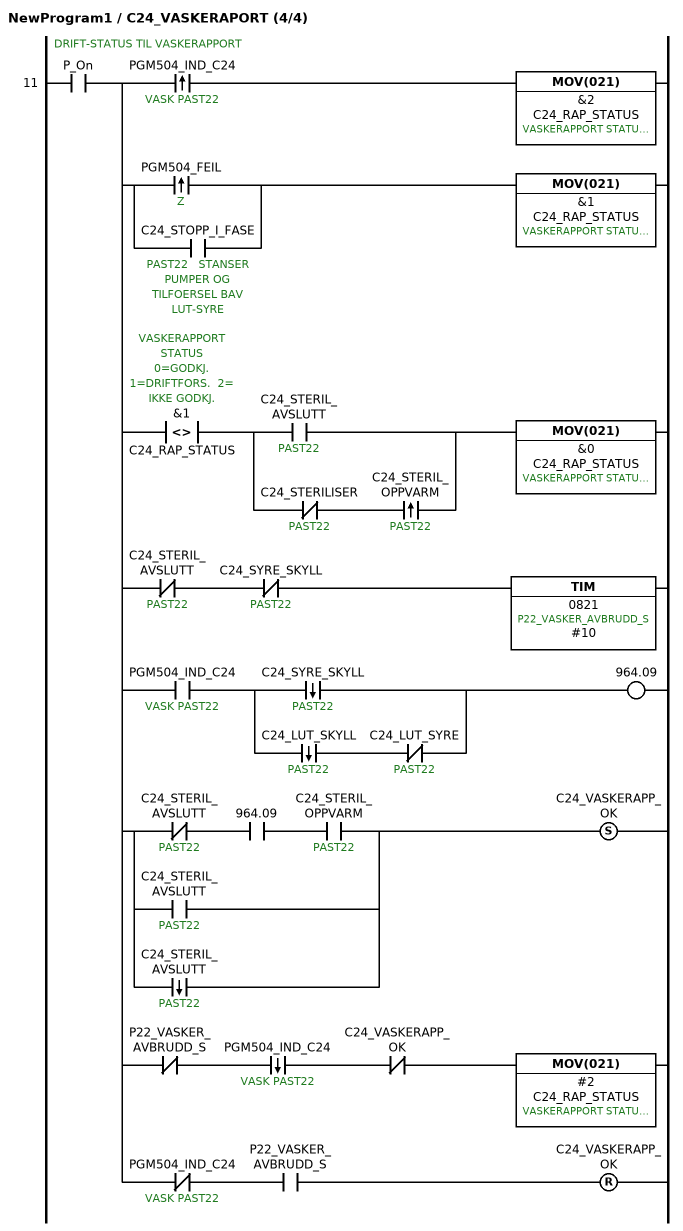
; rung 11: DRIFT-STATUS TIL VASKERAPPORT
LD P_On
OUT TR0
@AND PGM504_IND_C24  ; VASK PAST22
MOV(021) &2 C24_RAP_STATUS  ; VASKERAPPORT STATUS          0=GODKJ.  1=DRIFTFORS.  2= IKKE GODKJ.
LD TR0
@LD PGM504_FEIL  ; Z
OR C24_STOPP_I_FASE  ; PAST22   STANSER PUMPER OG TILFOERSEL BAV LUT-SYRE
ANDLD
MOV(021) &1 C24_RAP_STATUS  ; VASKERAPPORT STATUS          0=GODKJ.  1=DRIFTFORS.  2= IKKE GODKJ.
LD TR0
AND<>(305) &1 C24_RAP_STATUS  ; VASKERAPPORT STATUS          0=GODKJ.  1=DRIFTFORS.  2= IKKE GODKJ.
LD C24_STERIL_AVSLUTT  ; PAST22
LDNOT C24_STERILISER  ; PAST22
@AND C24_STERIL_OPPVARM  ; PAST22
ORLD
ANDLD
MOV(021) &0 C24_RAP_STATUS  ; VASKERAPPORT STATUS          0=GODKJ.  1=DRIFTFORS.  2= IKKE GODKJ.
LD TR0
ANDNOT C24_STERIL_AVSLUTT  ; PAST22
ANDNOT C24_SYRE_SKYLL  ; PAST22
TIM 0821 #10  ; P22_VASKER_AVBRUDD_S
LD TR0
AND PGM504_IND_C24  ; VASK PAST22
%LD C24_SYRE_SKYLL  ; PAST22
%LD C24_LUT_SKYLL  ; PAST22
ANDNOT C24_LUT_SYRE  ; PAST22
ORLD
ANDLD
OUT 964.09
LD TR0
LDNOT C24_STERIL_AVSLUTT  ; PAST22
AND 964.09
AND C24_STERIL_OPPVARM  ; PAST22
OR C24_STERIL_AVSLUTT  ; PAST22
%OR C24_STERIL_AVSLUTT  ; PAST22
ANDLD
SET C24_VASKERAPP_OK
LD TR0
ANDNOT P22_VASKER_AVBRUDD_S
%AND PGM504_IND_C24  ; VASK PAST22
ANDNOT C24_VASKERAPP_OK
MOV(021) #2 C24_RAP_STATUS  ; VASKERAPPORT STATUS          0=GODKJ.  1=DRIFTFORS.  2= IKKE GODKJ.
LD TR0
ANDNOT PGM504_IND_C24  ; VASK PAST22
AND P22_VASKER_AVBRUDD_S
RSET C24_VASKERAPP_OK
; rung 12: Ingen_kommentar_funnet

### Section C25_FUNKSJONER

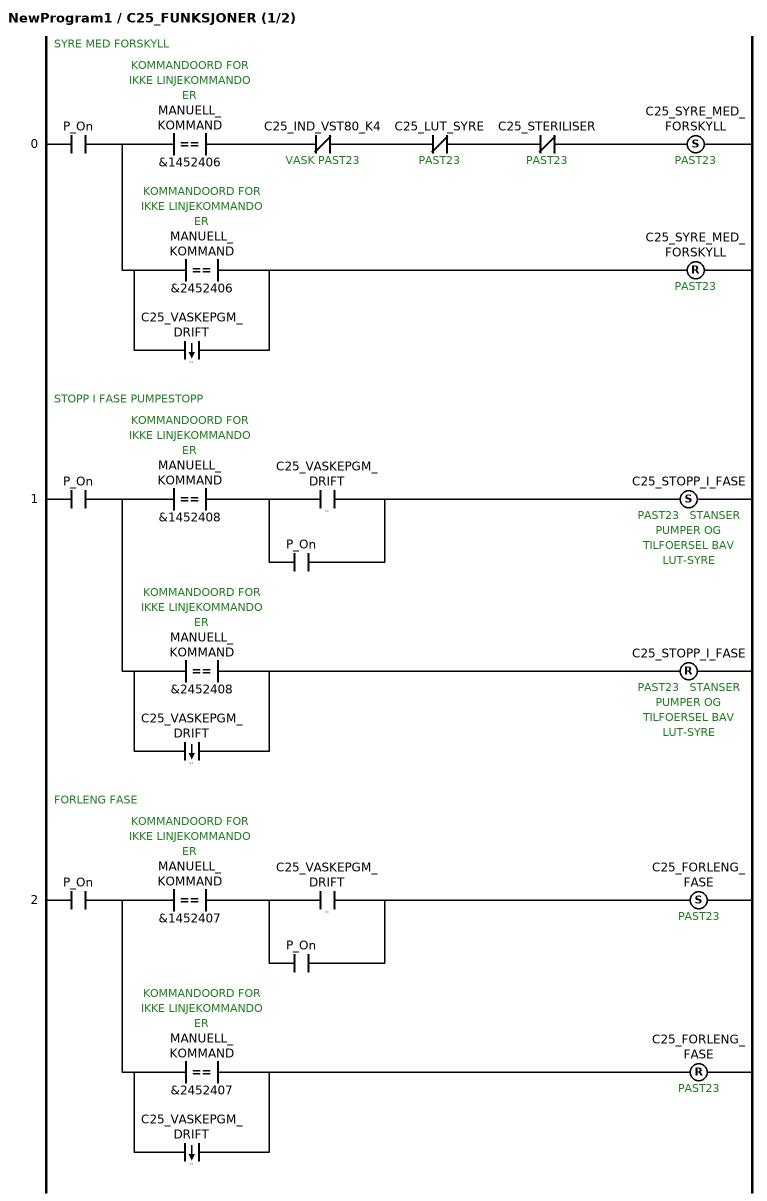
; rung 0: SYRE MED FORSKYLL
LD P_On
OUT TR0
AND=L(301) MANUELL_KOMMAND &1452406  ; KOMMANDOORD FOR IKKE LINJEKOMMANDOER
ANDNOT C25_IND_VST80_K4  ; VASK PAST23
ANDNOT C25_LUT_SYRE  ; PAST23
ANDNOT C25_STERILISER  ; PAST23
SET C25_SYRE_MED_FORSKYLL  ; PAST23
LD TR0
LD=L(301) MANUELL_KOMMAND &2452406  ; KOMMANDOORD FOR IKKE LINJEKOMMANDOER
%OR C25_VASKEPGM_DRIFT  ; ¨
ANDLD
RSET C25_SYRE_MED_FORSKYLL  ; PAST23
; rung 1: STOPP I FASE PUMPESTOPP
LD P_On
OUT TR0
AND=L(301) MANUELL_KOMMAND &1452408  ; KOMMANDOORD FOR IKKE LINJEKOMMANDOER
LD C25_VASKEPGM_DRIFT  ; ¨
OR P_On
ANDLD
SET C25_STOPP_I_FASE  ; PAST23   STANSER PUMPER OG TILFOERSEL BAV LUT-SYRE
LD TR0
LD=L(301) MANUELL_KOMMAND &2452408  ; KOMMANDOORD FOR IKKE LINJEKOMMANDOER
%OR C25_VASKEPGM_DRIFT  ; ¨
ANDLD
RSET C25_STOPP_I_FASE  ; PAST23   STANSER PUMPER OG TILFOERSEL BAV LUT-SYRE
; rung 2: FORLENG FASE
LD P_On
OUT TR0
AND=L(301) MANUELL_KOMMAND &1452407  ; KOMMANDOORD FOR IKKE LINJEKOMMANDOER
LD C25_VASKEPGM_DRIFT  ; ¨
OR P_On
ANDLD
SET C25_FORLENG_FASE  ; PAST23
LD TR0
LD=L(301) MANUELL_KOMMAND &2452407  ; KOMMANDOORD FOR IKKE LINJEKOMMANDOER
%OR C25_VASKEPGM_DRIFT  ; ¨
ANDLD
RSET C25_FORLENG_FASE  ; PAST23

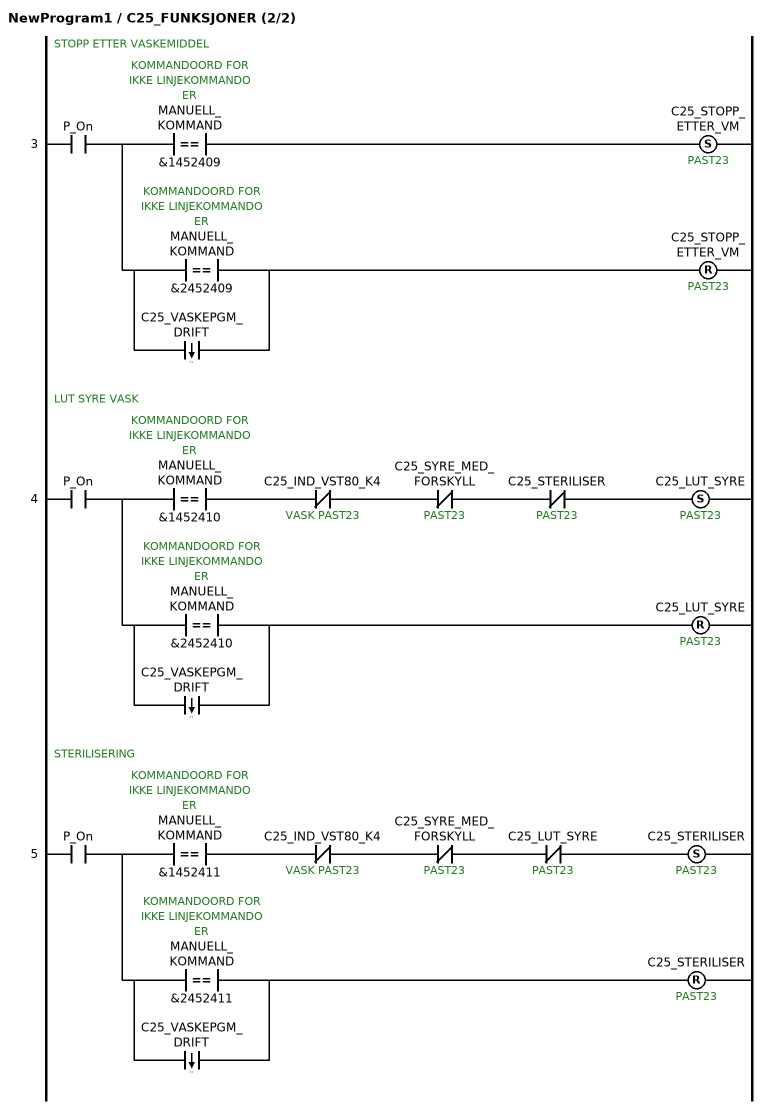
; rung 3: STOPP ETTER VASKEMIDDEL
LD P_On
OUT TR0
AND=L(301) MANUELL_KOMMAND &1452409  ; KOMMANDOORD FOR IKKE LINJEKOMMANDOER
SET C25_STOPP_ETTER_VM  ; PAST23
LD TR0
LD=L(301) MANUELL_KOMMAND &2452409  ; KOMMANDOORD FOR IKKE LINJEKOMMANDOER
%OR C25_VASKEPGM_DRIFT  ; ¨
ANDLD
RSET C25_STOPP_ETTER_VM  ; PAST23
; rung 4: LUT SYRE VASK
LD P_On
OUT TR0
AND=L(301) MANUELL_KOMMAND &1452410  ; KOMMANDOORD FOR IKKE LINJEKOMMANDOER
ANDNOT C25_IND_VST80_K4  ; VASK PAST23
ANDNOT C25_SYRE_MED_FORSKYLL  ; PAST23
ANDNOT C25_STERILISER  ; PAST23
SET C25_LUT_SYRE  ; PAST23
LD TR0
LD=L(301) MANUELL_KOMMAND &2452410  ; KOMMANDOORD FOR IKKE LINJEKOMMANDOER
%OR C25_VASKEPGM_DRIFT  ; ¨
ANDLD
RSET C25_LUT_SYRE  ; PAST23
; rung 5: STERILISERING
LD P_On
OUT TR0
AND=L(301) MANUELL_KOMMAND &1452411  ; KOMMANDOORD FOR IKKE LINJEKOMMANDOER
ANDNOT C25_IND_VST80_K4  ; VASK PAST23
ANDNOT C25_SYRE_MED_FORSKYLL  ; PAST23
ANDNOT C25_LUT_SYRE  ; PAST23
SET C25_STERILISER  ; PAST23
LD TR0
LD=L(301) MANUELL_KOMMAND &2452411  ; KOMMANDOORD FOR IKKE LINJEKOMMANDOER
%OR C25_VASKEPGM_DRIFT  ; ¨
ANDLD
RSET C25_STERILISER  ; PAST23
; rung 6: Ingen_kommentar_funnet

### Section VST80_C25_TRINN

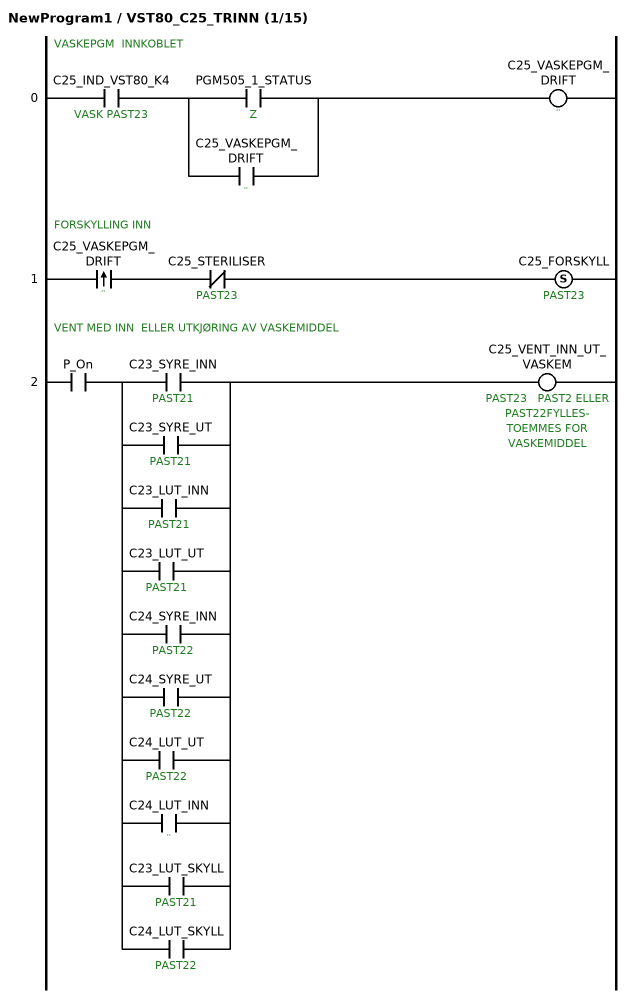
; rung 0: VASKEPGM  INNKOBLET
LD C25_IND_VST80_K4  ; VASK PAST23
LD PGM505_1_STATUS  ; Z
OR C25_VASKEPGM_DRIFT  ; ¨
ANDLD
OUT C25_VASKEPGM_DRIFT  ; ¨
; rung 1: FORSKYLLING INN
@LD C25_VASKEPGM_DRIFT  ; ¨
ANDNOT C25_STERILISER  ; PAST23
SET C25_FORSKYLL  ; PAST23
; rung 2: VENT MED INN  ELLER UTKJØRING AV VASKEMIDDEL
LD P_On
LD C23_SYRE_INN  ; PAST21
OR C23_SYRE_UT  ; PAST21
OR C23_LUT_INN  ; PAST21
OR C23_LUT_UT  ; PAST21
OR C24_SYRE_INN  ; PAST22
OR C24_SYRE_UT  ; PAST22
OR C24_LUT_UT  ; PAST22
OR C24_LUT_INN  ; ¨
OR C23_LUT_SKYLL  ; PAST21
OR C24_LUT_SKYLL  ; PAST22
ANDLD
OUT C25_VENT_INN_UT_VASKEM  ; PAST23   PAST2 ELLER PAST22FYLLES-TOEMMES FOR VASKEMIDDEL

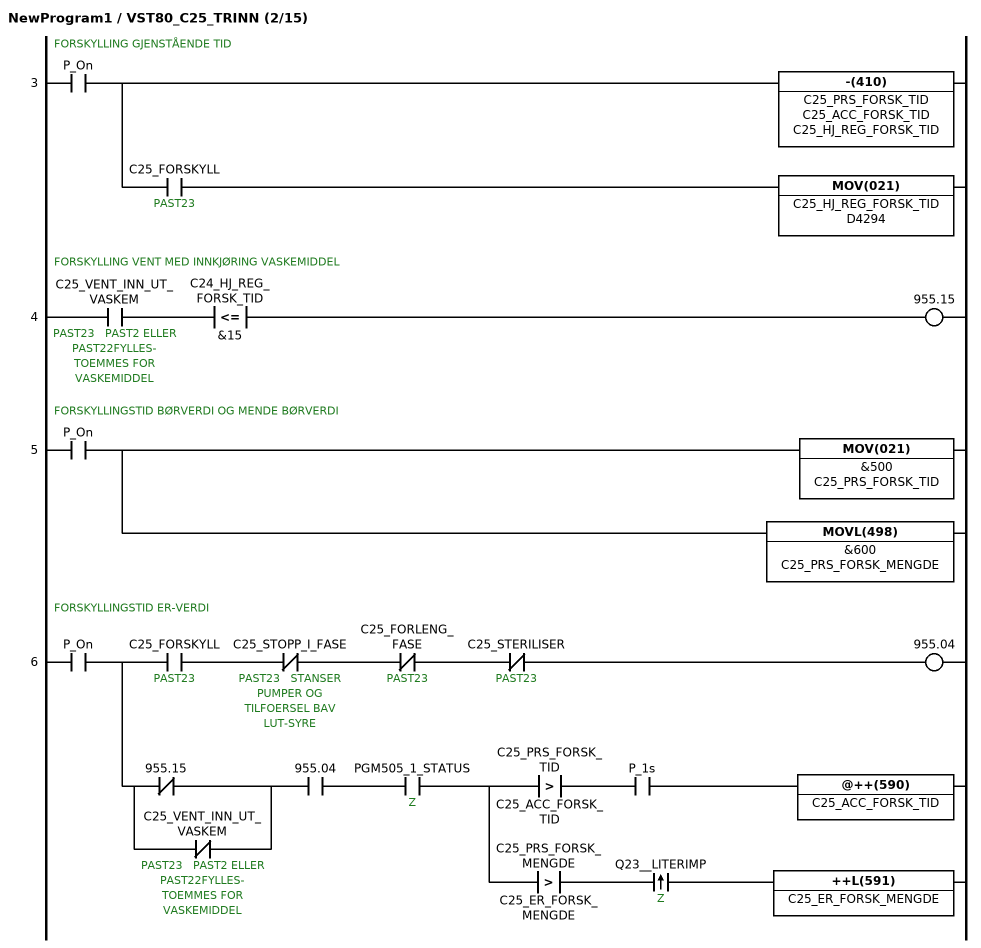
; rung 3: FORSKYLLING GJENSTÅENDE TID
LD P_On
-(410) C25_PRS_FORSK_TID C25_ACC_FORSK_TID C25_HJ_REG_FORSK_TID
AND C25_FORSKYLL  ; PAST23
MOV(021) C25_HJ_REG_FORSK_TID D4294
; rung 4: FORSKYLLING VENT MED INNKJØRING VASKEMIDDEL
LD C25_VENT_INN_UT_VASKEM  ; PAST23   PAST2 ELLER PAST22FYLLES-TOEMMES FOR VASKEMIDDEL
AND<=(315) C24_HJ_REG_FORSK_TID &15
OUT 955.15
; rung 5: FORSKYLLINGSTID BØRVERDI OG MENDE BØRVERDI
LD P_On
MOV(021) &500 C25_PRS_FORSK_TID
MOVL(498) &600 C25_PRS_FORSK_MENGDE
; rung 6: FORSKYLLINGSTID ER-VERDI
LD P_On
OUT TR0
AND C25_FORSKYLL  ; PAST23
ANDNOT C25_STOPP_I_FASE  ; PAST23   STANSER PUMPER OG TILFOERSEL BAV LUT-SYRE
ANDNOT C25_FORLENG_FASE  ; PAST23
ANDNOT C25_STERILISER  ; PAST23
OUT 955.04
LD TR0
LDNOT 955.15
ORNOT C25_VENT_INN_UT_VASKEM  ; PAST23   PAST2 ELLER PAST22FYLLES-TOEMMES FOR VASKEMIDDEL
ANDLD
AND 955.04
AND PGM505_1_STATUS  ; Z
OUT TR0
AND>(320) C25_PRS_FORSK_TID C25_ACC_FORSK_TID
AND P_1s
@++(590) C25_ACC_FORSK_TID
LD TR0
AND>(320) C25_PRS_FORSK_MENGDE C25_ER_FORSK_MENGDE
@AND Q23__LITERIMP  ; Z
++L(591) C25_ER_FORSK_MENGDE

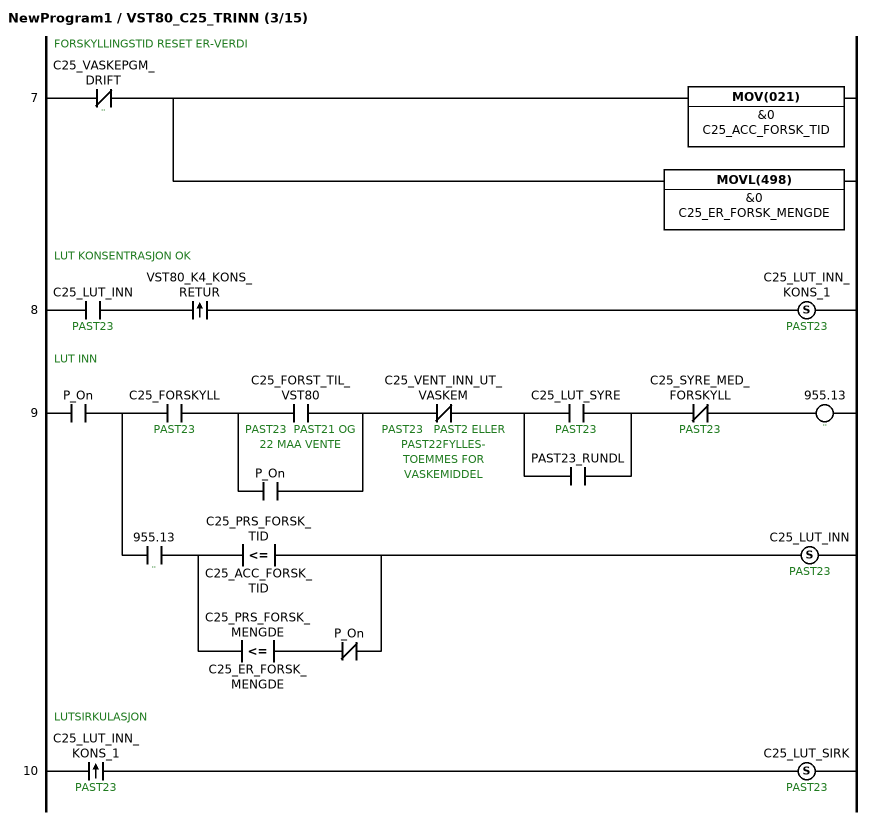
; rung 7: FORSKYLLINGSTID RESET ER-VERDI
LDNOT C25_VASKEPGM_DRIFT  ; ¨
MOV(021) &0 C25_ACC_FORSK_TID
MOVL(498) &0 C25_ER_FORSK_MENGDE
; rung 8: LUT KONSENTRASJON OK
LD C25_LUT_INN  ; PAST23
@AND VST80_K4_KONS_RETUR
SET C25_LUT_INN_KONS_1  ; PAST23
; rung 9: LUT INN
LD P_On
OUT TR0
AND C25_FORSKYLL  ; PAST23
LD C25_FORST_TIL_VST80  ; PAST23  PAST21 OG 22 MAA VENTE
OR P_On
ANDLD
ANDNOT C25_VENT_INN_UT_VASKEM  ; PAST23   PAST2 ELLER PAST22FYLLES-TOEMMES FOR VASKEMIDDEL
LD C25_LUT_SYRE  ; PAST23
OR PAST23_RUNDL
ANDLD
ANDNOT C25_SYRE_MED_FORSKYLL  ; PAST23
OUT 955.13  ; ¨
LD TR0
AND 955.13  ; ¨
LD<=(315) C25_PRS_FORSK_TID C25_ACC_FORSK_TID
LD<=L(316) C25_PRS_FORSK_MENGDE C25_ER_FORSK_MENGDE
ANDNOT P_On
ORLD
ANDLD
SET C25_LUT_INN  ; PAST23
; rung 10: LUTSIRKULASJON
@LD C25_LUT_INN_KONS_1  ; PAST23
SET C25_LUT_SIRK  ; PAST23

